// SIMATIC S7-200 project (STEP 7-Micro/WIN), CPU 224 REL 02.01

ORGANIZATION_BLOCK MAIN:OB1
TITLE=PROGRAM COMMENTS
BEGIN
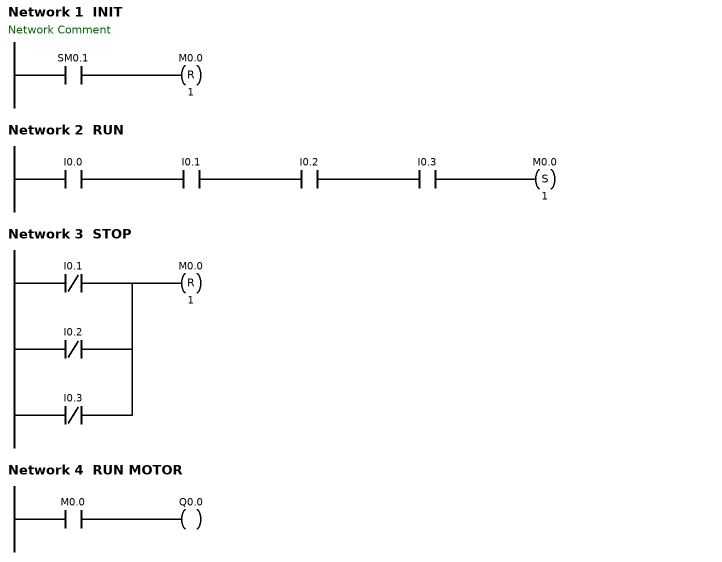
Network 1 // INIT
// Network Comment
LD     SM0.1
R      M0.0, 1
Network 2 // RUN
LD     I0.0
A      I0.1
A      I0.2
A      I0.3
S      M0.0, 1
Network 3 // STOP
LDN    I0.1
ON     I0.2
ON     I0.3
R      M0.0, 1
Network 4 // RUN MOTOR
LD     M0.0
=      Q0.0
END_ORGANIZATION_BLOCK
